KUKA KRL program: S_Zellenbereich.src, S_Zellenbereich.dat

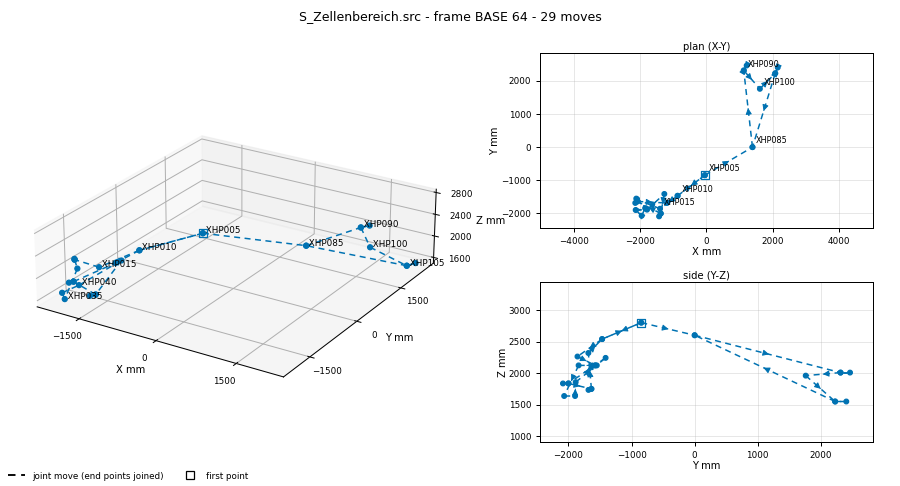
[picture p0: tool path of S_Zellenbereich.src in frame BASE 64, 29 of 31 moves have a stored position in this frame; points joined in program order, loops and branches not executed]
--- S_Zellenbereich.src ---
&ACCESS RVP
&REL 85
&COMMENT DAI_H_SOP_ZELLENBEREICH
&PARAM EDITMASK = DAI
&PARAM TEMPLATE = C:\KRC\roboter\template\vg_appl
&PARAM DISKPATH = KRC:\R1\H_Prog\DAI_SOP
DEF S_Zellenbereich( )
;FOLD INI;%{PE}
  ;FOLD BASISTECH INI
    GLOBAL INTERRUPT DECL 3 WHEN $STOPMESS==TRUE DO IR_STOPM ( )
    INTERRUPT ON 3
    BAS (#INITMOV,0 )
  ;ENDFOLD (BASISTECH INI)
  ;FOLD USER INI
    ;Make your modifications here
  ;ENDFOLD (USER INI)
;ENDFOLD (INI)
;FOLD ; Anlagenbezeichn: HC53_C    Stations-Nr: 060RB_100;%{PE}
;FOLD Parameters ;%{h}
;Params IlfProvider=kukaroboter.basistech.inlineforms.comments.comment; Kuka.Content=Anlagenbezeichn: HC53_C    Stations-Nr: 060RB_100
;ENDFOLD
;ENDFOLD
;FOLD ; Stand / Version: V1.0;%{PE}
;FOLD Parameters ;%{h}
;Params IlfProvider=kukaroboter.basistech.inlineforms.comments.comment; Kuka.Content=Stand / Version: V1.0
;ENDFOLD
;ENDFOLD
;FOLD ; Name Bearbeiter: EBZ-AE;%{PE}
;FOLD Parameters ;%{h}
;Params IlfProvider=kukaroboter.basistech.inlineforms.comments.comment; Kuka.Content=Name Bearbeiter: EBZ-AE
;ENDFOLD
;ENDFOLD
;FOLD ; Translator Version:29.01.2024 - Version 15.08;%{PE}
;FOLD Parameters ;%{h}
;Params IlfProvider=kukaroboter.basistech.inlineforms.comments.comment; Kuka.Content=Translator Version:29.01.2024 - Version 15.08
;ENDFOLD
;ENDFOLD

REPEAT
;FOLD MSG_T1
MSG_SHOW("DAI_H_SOP",#quit,999,"dai_h_sop_ok_0")
;ENDFOLD

; ***************************************
; A C H T U N G !!! Nur in $T1 abfahren
; ***************************************
UNTIL $T1 == TRUE

; ***************************************
; Pruefende Waende 4
;----------------------------------------
; Erreichbarkeit zum pruefen von P2/P3 nicht
; vorhanden.
;FOLD WAIT FOR ( IN 1026 'Vordefinierter Eingang immer ruckgesetzt.' )  ;%{PE}
;FOLD Parameters ;%{h}
;Params IlfProvider=kukaroboter.basistech.inlineforms.logics.waitfor; Kuka.WaitLogicTerm1=None; Kuka.WaitForNot1=False; Kuka.WaitLogicOp2.Term1=None; Kuka.WaitForNot2.Term1=False; Kuka.WaitForSysVar2.Term1=IN; Kuka.WaitForIndex2.Term1=1026; Kuka.WaitForIndexName2.Term1=Vordefinierter Eingang immer ruckgesetzt.; Kuka.WaitForTermNumbers=1; Kuka.WaitForOpNumbers=2; Kuka.WaitForCont=False
;ENDFOLD
WAIT FOR  ( $IN[1026] )
;ENDFOLD


;FOLD ; This program has been cleaned by KANERT_Makro. High risk of crash!!! Check the program carefully before deleting this comment. ;%{PE}
;FOLD Parameters ;%{h}
;Params IlfProvider=kukaroboter.basistech.inlineforms.comments.comment; Kuka.Content=This program has been cleaned by KANERT_Makro. High risk of crash!!! Check the program carefully before deleting this comment.
;ENDFOLD
WAIT FOR FALSE
;ENDFOLD
; ***************************************
;FOLD PTP HOME Vel=100 % DEFAULT;%{PE}
;FOLD Parameters ;%{h}
;Params IlfProvider=kukaroboter.basistech.inlineforms.movement.old; Kuka.IsGlobalPoint=False; Kuka.PointName=HOME; Kuka.BlendingEnabled=False; Kuka.MoveDataPtpName=DEFAULT; Kuka.VelocityPtp=100; Kuka.CurrentCDSetIndex=0; Kuka.MovementParameterFieldEnabled=True; IlfCommand=PTP
;ENDFOLD
$BWDSTART = FALSE
PDAT_ACT = PDEFAULT
FDAT_ACT = FHOME
BAS(#PTP_PARAMS, 100.0)
SET_CD_PARAMS (0)
PTP XHOME
;ENDFOLD

;Dynamische Pruefung Teil vorhanden
;FOLD PartPresent.CheckOff #1:5277, #2:5278, #3:1025, #4:1025, #5:1025, #6:1025, Bounce Time:100, Constant: Yes;%{PE}%
CheckPartPresent(5277,5278,1025,1025,1025,1025,100, True,FALSE)
;ENDFOLD

;Greifer-Ventile betatigen/pruefen
;FOLD DAI_GripValveCheck.Valve2 State:Fixierstift Ausfahren Gs, 060GRH101-QM1;%{PE}%
CheckValveState(2,1)
;ENDFOLD
;FOLD DAI_GripValveCheck.Valve3 State:Spanner Oeffnen Gs, 060GRH101-QM2;%{PE}%
CheckValveState(3,1)
;ENDFOLD
;FOLD DAI_GripValveCheck.Valve4 State:Spanner Oeffnen Gs, 060GRH101-QM3;%{PE}%
CheckValveState(4,1)
;ENDFOLD

;FOLD PTP HP005 Vel=100 % PDAT1 Tool[64]:Zero Base[64]:Zero ;%{PE}
;FOLD Parameters ;%{h}
;Params IlfProvider=kukaroboter.basistech.inlineforms.movement.old; Kuka.IsGlobalPoint=False; Kuka.PointName=HP005; Kuka.BlendingEnabled=False; Kuka.MoveDataPtpName=PDAT1; Kuka.VelocityPtp=100; Kuka.CurrentCDSetIndex=0; Kuka.MovementParameterFieldEnabled=True; IlfCommand=PTP
;ENDFOLD
$BWDSTART = FALSE
PDAT_ACT = PPDAT1
FDAT_ACT = FHP005
BAS(#PTP_PARAMS, 100.0)
SET_CD_PARAMS (0)
PTP XHP005
;ENDFOLD
;FOLD PTP HP010 Vel=100 % PDAT2 Tool[64]:Zero Base[64]:Zero ;%{PE}
;FOLD Parameters ;%{h}
;Params IlfProvider=kukaroboter.basistech.inlineforms.movement.old; Kuka.IsGlobalPoint=False; Kuka.PointName=HP010; Kuka.BlendingEnabled=False; Kuka.MoveDataPtpName=PDAT2; Kuka.VelocityPtp=100; Kuka.CurrentCDSetIndex=0; Kuka.MovementParameterFieldEnabled=True; IlfCommand=PTP
;ENDFOLD
$BWDSTART = FALSE
PDAT_ACT = PPDAT2
FDAT_ACT = FHP010
BAS(#PTP_PARAMS, 100.0)
SET_CD_PARAMS (0)
PTP XHP010
;ENDFOLD
;FOLD PTP HP015 Vel=100 % PDAT3 Tool[64]:Zero Base[64]:Zero ;%{PE}
;FOLD Parameters ;%{h}
;Params IlfProvider=kukaroboter.basistech.inlineforms.movement.old; Kuka.IsGlobalPoint=False; Kuka.PointName=HP015; Kuka.BlendingEnabled=False; Kuka.MoveDataPtpName=PDAT3; Kuka.VelocityPtp=100; Kuka.CurrentCDSetIndex=0; Kuka.MovementParameterFieldEnabled=True; IlfCommand=PTP
;ENDFOLD
$BWDSTART = FALSE
PDAT_ACT = PPDAT3
FDAT_ACT = FHP015
BAS(#PTP_PARAMS, 100.0)
SET_CD_PARAMS (0)
PTP XHP015
;ENDFOLD
;FOLD PTP HP020 Vel=100 % PDAT4 Tool[64]:Zero Base[64]:Zero;%{PE}
;FOLD Parameters ;%{h}
;Params IlfProvider=kukaroboter.basistech.inlineforms.movement.old; Kuka.IsGlobalPoint=False; Kuka.PointName=HP020; Kuka.BlendingEnabled=False; Kuka.MoveDataPtpName=PDAT4; Kuka.VelocityPtp=100; Kuka.CurrentCDSetIndex=0; Kuka.MovementParameterFieldEnabled=True; IlfCommand=PTP
;ENDFOLD
$BWDSTART = FALSE
PDAT_ACT = PPDAT4
FDAT_ACT = FHP020
BAS(#PTP_PARAMS, 100.0)
SET_CD_PARAMS (0)
PTP XHP020
;ENDFOLD

; Pruefung Raum P1n
;FOLD PTP LPruef01_Zellenbereich Vel=100 % PDAT5 Tool[64]:Zero Base[64]:Zero ;%{PE}
;FOLD Parameters ;%{h}
;Params IlfProvider=kukaroboter.basistech.inlineforms.movement.old; Kuka.IsGlobalPoint=False; Kuka.PointName=LPruef01_Zellenbereich; Kuka.BlendingEnabled=False; Kuka.MoveDataPtpName=PDAT5; Kuka.VelocityPtp=100; Kuka.CurrentCDSetIndex=0; Kuka.MovementParameterFieldEnabled=True; IlfCommand=PTP
;ENDFOLD
$BWDSTART = FALSE
PDAT_ACT = PPDAT5
FDAT_ACT = FLPruef01_Zellenbereich
BAS(#PTP_PARAMS, 100.0)
SET_CD_PARAMS (0)
PTP XLPruef01_Zellenbereich
;ENDFOLD
;FOLD PTP HP025 Vel=100 % PDAT6 Tool[64]:Zero Base[64]:Zero ;%{PE}
;FOLD Parameters ;%{h}
;Params IlfProvider=kukaroboter.basistech.inlineforms.movement.old; Kuka.IsGlobalPoint=False; Kuka.PointName=HP025; Kuka.BlendingEnabled=False; Kuka.MoveDataPtpName=PDAT6; Kuka.VelocityPtp=100; Kuka.CurrentCDSetIndex=0; Kuka.MovementParameterFieldEnabled=True; IlfCommand=PTP
;ENDFOLD
$BWDSTART = FALSE
PDAT_ACT = PPDAT6
FDAT_ACT = FHP025
BAS(#PTP_PARAMS, 100.0)
SET_CD_PARAMS (0)
PTP XHP025
;ENDFOLD
;FOLD PTP HP030 Vel=100 % PDAT7 Tool[64]:Zero Base[64]:Zero;%{PE}
;FOLD Parameters ;%{h}
;Params IlfProvider=kukaroboter.basistech.inlineforms.movement.old; Kuka.IsGlobalPoint=False; Kuka.PointName=HP030; Kuka.BlendingEnabled=False; Kuka.MoveDataPtpName=PDAT7; Kuka.VelocityPtp=100; Kuka.CurrentCDSetIndex=0; Kuka.MovementParameterFieldEnabled=True; IlfCommand=PTP
;ENDFOLD
$BWDSTART = FALSE
PDAT_ACT = PPDAT7
FDAT_ACT = FHP030
BAS(#PTP_PARAMS, 100.0)
SET_CD_PARAMS (0)
PTP XHP030
;ENDFOLD
;FOLD PTP HP035 Vel=100 % PDAT8 Tool[64]:Zero Base[64]:Zero;%{PE}
;FOLD Parameters ;%{h}
;Params IlfProvider=kukaroboter.basistech.inlineforms.movement.old; Kuka.IsGlobalPoint=False; Kuka.PointName=HP035; Kuka.BlendingEnabled=False; Kuka.MoveDataPtpName=PDAT8; Kuka.VelocityPtp=100; Kuka.CurrentCDSetIndex=0; Kuka.MovementParameterFieldEnabled=True; IlfCommand=PTP
;ENDFOLD
$BWDSTART = FALSE
PDAT_ACT = PPDAT8
FDAT_ACT = FHP035
BAS(#PTP_PARAMS, 100.0)
SET_CD_PARAMS (0)
PTP XHP035
;ENDFOLD

; Pruefung Raum P2
;FOLD PTP LPruef02_Zellenbereich Vel=100 % PDAT9 Tool[64]:Zero Base[64]:Zero ;%{PE}
;FOLD Parameters ;%{h}
;Params IlfProvider=kukaroboter.basistech.inlineforms.movement.old; Kuka.IsGlobalPoint=False; Kuka.PointName=LPruef02_Zellenbereich; Kuka.BlendingEnabled=False; Kuka.MoveDataPtpName=PDAT9; Kuka.VelocityPtp=100; Kuka.CurrentCDSetIndex=0; Kuka.MovementParameterFieldEnabled=True; IlfCommand=PTP
;ENDFOLD
$BWDSTART = FALSE
PDAT_ACT = PPDAT9
FDAT_ACT = FLPruef02_Zellenbereich
BAS(#PTP_PARAMS, 100.0)
SET_CD_PARAMS (0)
PTP XLPruef02_Zellenbereich
;ENDFOLD
;FOLD PTP HP040 Vel=100 % PDAT10 Tool[64]:Zero Base[64]:Zero ;%{PE}
;FOLD Parameters ;%{h}
;Params IlfProvider=kukaroboter.basistech.inlineforms.movement.old; Kuka.IsGlobalPoint=False; Kuka.PointName=HP040; Kuka.BlendingEnabled=False; Kuka.MoveDataPtpName=PDAT10; Kuka.VelocityPtp=100; Kuka.CurrentCDSetIndex=0; Kuka.MovementParameterFieldEnabled=True; IlfCommand=PTP
;ENDFOLD
$BWDSTART = FALSE
PDAT_ACT = PPDAT10
FDAT_ACT = FHP040
BAS(#PTP_PARAMS, 100.0)
SET_CD_PARAMS (0)
PTP XHP040
;ENDFOLD
;FOLD PTP HP045 Vel=100 % PDAT11 Tool[64]:Zero Base[64]:Zero ;%{PE}
;FOLD Parameters ;%{h}
;Params IlfProvider=kukaroboter.basistech.inlineforms.movement.old; Kuka.IsGlobalPoint=False; Kuka.PointName=HP045; Kuka.BlendingEnabled=False; Kuka.MoveDataPtpName=PDAT11; Kuka.VelocityPtp=100; Kuka.CurrentCDSetIndex=0; Kuka.MovementParameterFieldEnabled=True; IlfCommand=PTP
;ENDFOLD
$BWDSTART = FALSE
PDAT_ACT = PPDAT11
FDAT_ACT = FHP045
BAS(#PTP_PARAMS, 100.0)
SET_CD_PARAMS (0)
PTP XHP045
;ENDFOLD
;FOLD PTP HP050 Vel=100 % PDAT12 Tool[64]:Zero Base[64]:Zero ;%{PE}
;FOLD Parameters ;%{h}
;Params IlfProvider=kukaroboter.basistech.inlineforms.movement.old; Kuka.IsGlobalPoint=False; Kuka.PointName=HP050; Kuka.BlendingEnabled=False; Kuka.MoveDataPtpName=PDAT12; Kuka.VelocityPtp=100; Kuka.CurrentCDSetIndex=0; Kuka.MovementParameterFieldEnabled=True; IlfCommand=PTP
;ENDFOLD
$BWDSTART = FALSE
PDAT_ACT = PPDAT12
FDAT_ACT = FHP050
BAS(#PTP_PARAMS, 100.0)
SET_CD_PARAMS (0)
PTP XHP050
;ENDFOLD

; Pruefung Raum P3
;FOLD PTP LPruef03_Zellenbereich Vel=100 % PDAT13 Tool[64]:Zero Base[64]:Zero ;%{PE}
;FOLD Parameters ;%{h}
;Params IlfProvider=kukaroboter.basistech.inlineforms.movement.old; Kuka.IsGlobalPoint=False; Kuka.PointName=LPruef03_Zellenbereich; Kuka.BlendingEnabled=False; Kuka.MoveDataPtpName=PDAT13; Kuka.VelocityPtp=100; Kuka.CurrentCDSetIndex=0; Kuka.MovementParameterFieldEnabled=True; IlfCommand=PTP
;ENDFOLD
$BWDSTART = FALSE
PDAT_ACT = PPDAT13
FDAT_ACT = FLPruef03_Zellenbereich
BAS(#PTP_PARAMS, 100.0)
SET_CD_PARAMS (0)
PTP XLPruef03_Zellenbereich
;ENDFOLD
;FOLD PTP HP055 Vel=100 % PDAT14 Tool[64]:Zero Base[64]:Zero ;%{PE}
;FOLD Parameters ;%{h}
;Params IlfProvider=kukaroboter.basistech.inlineforms.movement.old; Kuka.IsGlobalPoint=False; Kuka.PointName=HP055; Kuka.BlendingEnabled=False; Kuka.MoveDataPtpName=PDAT14; Kuka.VelocityPtp=100; Kuka.CurrentCDSetIndex=0; Kuka.MovementParameterFieldEnabled=True; IlfCommand=PTP
;ENDFOLD
$BWDSTART = FALSE
PDAT_ACT = PPDAT14
FDAT_ACT = FHP055
BAS(#PTP_PARAMS, 100.0)
SET_CD_PARAMS (0)
PTP XHP055
;ENDFOLD
;FOLD PTP HP060 Vel=100 % PDAT15 Tool[64]:Zero Base[64]:Zero ;%{PE}
;FOLD Parameters ;%{h}
;Params IlfProvider=kukaroboter.basistech.inlineforms.movement.old; Kuka.IsGlobalPoint=False; Kuka.PointName=HP060; Kuka.BlendingEnabled=False; Kuka.MoveDataPtpName=PDAT15; Kuka.VelocityPtp=100; Kuka.CurrentCDSetIndex=0; Kuka.MovementParameterFieldEnabled=True; IlfCommand=PTP
;ENDFOLD
$BWDSTART = FALSE
PDAT_ACT = PPDAT15
FDAT_ACT = FHP060
BAS(#PTP_PARAMS, 100.0)
SET_CD_PARAMS (0)
PTP XHP060
;ENDFOLD

; Pruefung Raum P4
;FOLD PTP LPruef04_Zellenbereich Vel=100 % PDAT16 Tool[64]:Zero Base[64]:Zero ;%{PE}
;FOLD Parameters ;%{h}
;Params IlfProvider=kukaroboter.basistech.inlineforms.movement.old; Kuka.IsGlobalPoint=False; Kuka.PointName=LPruef04_Zellenbereich; Kuka.BlendingEnabled=False; Kuka.MoveDataPtpName=PDAT16; Kuka.VelocityPtp=100; Kuka.CurrentCDSetIndex=0; Kuka.MovementParameterFieldEnabled=True; IlfCommand=PTP
;ENDFOLD
$BWDSTART = FALSE
PDAT_ACT = PPDAT16
FDAT_ACT = FLPruef04_Zellenbereich
BAS(#PTP_PARAMS, 100.0)
SET_CD_PARAMS (0)
PTP XLPruef04_Zellenbereich
;ENDFOLD
;FOLD PTP HP065 Vel=100 % PDAT17 Tool[64]:Zero Base[64]:Zero ;%{PE}
;FOLD Parameters ;%{h}
;Params IlfProvider=kukaroboter.basistech.inlineforms.movement.old; Kuka.IsGlobalPoint=False; Kuka.PointName=HP065; Kuka.BlendingEnabled=False; Kuka.MoveDataPtpName=PDAT17; Kuka.VelocityPtp=100; Kuka.CurrentCDSetIndex=0; Kuka.MovementParameterFieldEnabled=True; IlfCommand=PTP
;ENDFOLD
$BWDSTART = FALSE
PDAT_ACT = PPDAT17
FDAT_ACT = FHP065
BAS(#PTP_PARAMS, 100.0)
SET_CD_PARAMS (0)
PTP XHP065
;ENDFOLD
;FOLD PTP HP070 Vel=100 % PDAT18 Tool[64]:Zero Base[64]:Zero ;%{PE}
;FOLD Parameters ;%{h}
;Params IlfProvider=kukaroboter.basistech.inlineforms.movement.old; Kuka.IsGlobalPoint=False; Kuka.PointName=HP070; Kuka.BlendingEnabled=False; Kuka.MoveDataPtpName=PDAT18; Kuka.VelocityPtp=100; Kuka.CurrentCDSetIndex=0; Kuka.MovementParameterFieldEnabled=True; IlfCommand=PTP
;ENDFOLD
$BWDSTART = FALSE
PDAT_ACT = PPDAT18
FDAT_ACT = FHP070
BAS(#PTP_PARAMS, 100.0)
SET_CD_PARAMS (0)
PTP XHP070
;ENDFOLD
;FOLD PTP HP075 Vel=100 % PDAT19 Tool[64]:Zero Base[64]:Zero ;%{PE}
;FOLD Parameters ;%{h}
;Params IlfProvider=kukaroboter.basistech.inlineforms.movement.old; Kuka.IsGlobalPoint=False; Kuka.PointName=HP075; Kuka.BlendingEnabled=False; Kuka.MoveDataPtpName=PDAT19; Kuka.VelocityPtp=100; Kuka.CurrentCDSetIndex=0; Kuka.MovementParameterFieldEnabled=True; IlfCommand=PTP
;ENDFOLD
$BWDSTART = FALSE
PDAT_ACT = PPDAT19
FDAT_ACT = FHP075
BAS(#PTP_PARAMS, 100.0)
SET_CD_PARAMS (0)
PTP XHP075
;ENDFOLD
;FOLD PTP HP080 Vel=100 % PDAT20 Tool[64]:Zero Base[64]:Zero ;%{PE}
;FOLD Parameters ;%{h}
;Params IlfProvider=kukaroboter.basistech.inlineforms.movement.old; Kuka.IsGlobalPoint=False; Kuka.PointName=HP080; Kuka.BlendingEnabled=False; Kuka.MoveDataPtpName=PDAT20; Kuka.VelocityPtp=100; Kuka.CurrentCDSetIndex=0; Kuka.MovementParameterFieldEnabled=True; IlfCommand=PTP
;ENDFOLD
$BWDSTART = FALSE
PDAT_ACT = PPDAT20
FDAT_ACT = FHP080
BAS(#PTP_PARAMS, 100.0)
SET_CD_PARAMS (0)
PTP XHP080
;ENDFOLD
;FOLD PTP HP085 Vel=100 % PDAT21 Tool[64]:Zero Base[64]:Zero ;%{PE}
;FOLD Parameters ;%{h}
;Params IlfProvider=kukaroboter.basistech.inlineforms.movement.old; Kuka.IsGlobalPoint=False; Kuka.PointName=HP085; Kuka.BlendingEnabled=False; Kuka.MoveDataPtpName=PDAT21; Kuka.VelocityPtp=100; Kuka.CurrentCDSetIndex=0; Kuka.MovementParameterFieldEnabled=True; IlfCommand=PTP
;ENDFOLD
$BWDSTART = FALSE
PDAT_ACT = PPDAT21
FDAT_ACT = FHP085
BAS(#PTP_PARAMS, 100.0)
SET_CD_PARAMS (0)
PTP XHP085
;ENDFOLD
;FOLD PTP HP090 Vel=100 % PDAT22 Tool[64]:Zero Base[64]:Zero;%{PE}
;FOLD Parameters ;%{h}
;Params IlfProvider=kukaroboter.basistech.inlineforms.movement.old; Kuka.IsGlobalPoint=False; Kuka.PointName=HP090; Kuka.BlendingEnabled=False; Kuka.MoveDataPtpName=PDAT22; Kuka.VelocityPtp=100; Kuka.CurrentCDSetIndex=0; Kuka.MovementParameterFieldEnabled=True; IlfCommand=PTP
;ENDFOLD
$BWDSTART = FALSE
PDAT_ACT = PPDAT22
FDAT_ACT = FHP090
BAS(#PTP_PARAMS, 100.0)
SET_CD_PARAMS (0)
PTP XHP090
;ENDFOLD

; Pruefung Raum P5
;FOLD PTP LPruef05_Zellenbereich Vel=100 % PDAT23 Tool[64]:Zero Base[64]:Zero ;%{PE}
;FOLD Parameters ;%{h}
;Params IlfProvider=kukaroboter.basistech.inlineforms.movement.old; Kuka.IsGlobalPoint=False; Kuka.PointName=LPruef05_Zellenbereich; Kuka.BlendingEnabled=False; Kuka.MoveDataPtpName=PDAT23; Kuka.VelocityPtp=100; Kuka.CurrentCDSetIndex=0; Kuka.MovementParameterFieldEnabled=True; IlfCommand=PTP
;ENDFOLD
$BWDSTART = FALSE
PDAT_ACT = PPDAT23
FDAT_ACT = FLPruef05_Zellenbereich
BAS(#PTP_PARAMS, 100.0)
SET_CD_PARAMS (0)
PTP XLPruef05_Zellenbereich
;ENDFOLD
;FOLD PTP HP095 Vel=100 % PDAT24 Tool[64]:Zero Base[64]:Zero ;%{PE}
;FOLD Parameters ;%{h}
;Params IlfProvider=kukaroboter.basistech.inlineforms.movement.old; Kuka.IsGlobalPoint=False; Kuka.PointName=HP095; Kuka.BlendingEnabled=False; Kuka.MoveDataPtpName=PDAT24; Kuka.VelocityPtp=100; Kuka.CurrentCDSetIndex=0; Kuka.MovementParameterFieldEnabled=True; IlfCommand=PTP
;ENDFOLD
$BWDSTART = FALSE
PDAT_ACT = PPDAT24
FDAT_ACT = FHP095
BAS(#PTP_PARAMS, 100.0)
SET_CD_PARAMS (0)
PTP XHP095
;ENDFOLD
;FOLD PTP HP100 Vel=100 % PDAT25 Tool[64]:Zero Base[64]:Zero;%{PE}
;FOLD Parameters ;%{h}
;Params IlfProvider=kukaroboter.basistech.inlineforms.movement.old; Kuka.IsGlobalPoint=False; Kuka.PointName=HP100; Kuka.BlendingEnabled=False; Kuka.MoveDataPtpName=PDAT25; Kuka.VelocityPtp=100; Kuka.CurrentCDSetIndex=0; Kuka.MovementParameterFieldEnabled=True; IlfCommand=PTP
;ENDFOLD
$BWDSTART = FALSE
PDAT_ACT = PPDAT25
FDAT_ACT = FHP100
BAS(#PTP_PARAMS, 100.0)
SET_CD_PARAMS (0)
PTP XHP100
;ENDFOLD
;FOLD PTP HP105 Vel=100 % PDAT26 Tool[64]:Zero Base[64]:Zero;%{PE}
;FOLD Parameters ;%{h}
;Params IlfProvider=kukaroboter.basistech.inlineforms.movement.old; Kuka.IsGlobalPoint=False; Kuka.PointName=HP105; Kuka.BlendingEnabled=False; Kuka.MoveDataPtpName=PDAT26; Kuka.VelocityPtp=100; Kuka.CurrentCDSetIndex=0; Kuka.MovementParameterFieldEnabled=True; IlfCommand=PTP
;ENDFOLD
$BWDSTART = FALSE
PDAT_ACT = PPDAT26
FDAT_ACT = FHP105
BAS(#PTP_PARAMS, 100.0)
SET_CD_PARAMS (0)
PTP XHP105
;ENDFOLD

; Pruefung Raum P6
;FOLD PTP LPruef06_Zellenbereich Vel=100 % PDAT27 Tool[64]:Zero Base[64]:Zero ;%{PE}
;FOLD Parameters ;%{h}
;Params IlfProvider=kukaroboter.basistech.inlineforms.movement.old; Kuka.IsGlobalPoint=False; Kuka.PointName=LPruef06_Zellenbereich; Kuka.BlendingEnabled=False; Kuka.MoveDataPtpName=PDAT27; Kuka.VelocityPtp=100; Kuka.CurrentCDSetIndex=0; Kuka.MovementParameterFieldEnabled=True; IlfCommand=PTP
;ENDFOLD
$BWDSTART = FALSE
PDAT_ACT = PPDAT27
FDAT_ACT = FLPruef06_Zellenbereich
BAS(#PTP_PARAMS, 100.0)
SET_CD_PARAMS (0)
PTP XLPruef06_Zellenbereich
;ENDFOLD
;FOLD PTP HP110 Vel=100 % PDAT28 Tool[64]:Zero Base[64]:Zero;%{PE}
;FOLD Parameters ;%{h}
;Params IlfProvider=kukaroboter.basistech.inlineforms.movement.old; Kuka.IsGlobalPoint=False; Kuka.PointName=HP110; Kuka.BlendingEnabled=False; Kuka.MoveDataPtpName=PDAT28; Kuka.VelocityPtp=100; Kuka.CurrentCDSetIndex=0; Kuka.MovementParameterFieldEnabled=True; IlfCommand=PTP
;ENDFOLD
$BWDSTART = FALSE
PDAT_ACT = PPDAT28
FDAT_ACT = FHP110
BAS(#PTP_PARAMS, 100.0)
SET_CD_PARAMS (0)
PTP XHP110
;ENDFOLD
;FOLD PTP HP115 Vel=100 % PDAT29 Tool[64]:Zero Base[64]:Zero;%{PE}
;FOLD Parameters ;%{h}
;Params IlfProvider=kukaroboter.basistech.inlineforms.movement.old; Kuka.IsGlobalPoint=False; Kuka.PointName=HP115; Kuka.BlendingEnabled=False; Kuka.MoveDataPtpName=PDAT29; Kuka.VelocityPtp=100; Kuka.CurrentCDSetIndex=0; Kuka.MovementParameterFieldEnabled=True; IlfCommand=PTP
;ENDFOLD
$BWDSTART = FALSE
PDAT_ACT = PPDAT29
FDAT_ACT = FHP115
BAS(#PTP_PARAMS, 100.0)
SET_CD_PARAMS (0)
PTP XHP115
;ENDFOLD

;FOLD PTP HOME Vel=100 % DEFAULT;%{PE}
;FOLD Parameters ;%{h}
;Params IlfProvider=kukaroboter.basistech.inlineforms.movement.old; Kuka.IsGlobalPoint=False; Kuka.PointName=HOME; Kuka.BlendingEnabled=False; Kuka.MoveDataPtpName=DEFAULT; Kuka.VelocityPtp=100; Kuka.CurrentCDSetIndex=0; Kuka.MovementParameterFieldEnabled=True; IlfCommand=PTP
;ENDFOLD
$BWDSTART = FALSE
PDAT_ACT = PDEFAULT
FDAT_ACT = FHOME
BAS(#PTP_PARAMS, 100.0)
SET_CD_PARAMS (0)
PTP XHOME
;ENDFOLD

;Collision detection - Off
;FOLD COLLDETECT Off ;%{PE}
;FOLD Parameters ;%{h}
;Params IlfProvider=kukaroboter.basistech.inlineforms.colldetect.off; CollDetect.Command=Off
;ENDFOLD
USE_CD_PARAMS(0)
;ENDFOLD
END

--- S_Zellenbereich.dat ---
&ACCESS RVO
&REL 86
&COMMENT DAI_H_SOP_ZELLENBEREICH
&PARAM EDITMASK = DAI
&PARAM TEMPLATE = C:\KRC\roboter\template\vg_appl
&PARAM DISKPATH = KRC:\R1\H_Prog\DAI_SOP
DEFDAT  S_ZELLENBEREICH
;FOLD EXTERNAL DECLARATIONS;%{PE}%MKUKATPBASIS,%CEXT,%VCOMMON,%P
;FOLD BASISTECH EXT;%{PE}%MKUKATPBASIS,%CEXT,%VEXT,%P
EXT  BAS (BAS_COMMAND  :IN,REAL  :IN )
DECL INT SUCCESS
;ENDFOLD (BASISTECH EXT)
;FOLD USER EXT;%{E}%MKUKATPUSER,%CEXT,%VEXT,%P
;Make your modifications here
;ENDFOLD (USER EXT)
;FOLD COLLISION
EXT  COLLSTOP (INT  :IN,INT  :IN )
;ENDFOLD  (Collision)
;ENDFOLD (EXTERNAL DECLERATIONS)
DECL BASIS_SUGG_T LAST_BASIS={POINT1[] "P0                      ",POINT2[] "P0                      ",CP_PARAMS[] "CPDAT0                  ",PTP_PARAMS[] "PDAT0                   ",CONT[] "                        ",CP_VEL[] "2.0                     ",PTP_VEL[] "100                     ",SYNC_PARAMS[] "SYNCDAT                 ",SPL_NAME[] "S0                      ",A_PARAMS[] "ADAT0                   "}
DECL MODULEPARAM_T LAST_TP_PARAMS={PARAMS[] "Kuka.PointName=LPruef11_Zellenbereich; Kuka.FrameData.base_no=64; Kuka.FrameData.tool_no=64; Kuka.FrameData.ipo_frame=#BASE; Kuka.FrameData.point2=; Kuka.isglobalpoint=False; Kuka.MoveDataPtpName=PDAT42; Kuka.MovementDataPdat.apo_mode=#CDIS; Kuka.MovementDataPdat.apo_dist=500; Kuka.MovementData.vel=100; Kuka.MovementData.acc=100; Kuka.MovementData.exax_ign=0; Kuka.VelocityPtp=100; Kuka.BlendingEnabled=False; Kuka.APXEnabled=False; Kuka.CurrentCDSetIndex=0"}

; E6POS Declarations
DECL E6POS XHP005={X -46.1297722,Y -846.191040,Z 2801.22607,A 172.487946,B -23.7688217,C -126.323227,S 18,T 10,E1 -351.691864,E2 0.0,E3 0.0,E4 0.0,E5 0.0,E6 0.0}
DECL E6POS XHP010={X -867.191101,Y -1466.68518,Z 2540.40723,A -152.699829,B -31.1417503,C -161.784149,S 18,T 10,E1 -164.100861,E2 0.0,E3 0.0,E4 0.0,E5 0.0,E6 0.0}
DECL E6POS XHP015={X -1396.02393,Y -1857.07593,Z 2264.14600,A -150.484390,B -25.5367279,C -163.976059,S 18,T 10,E1 21.3274384,E2 0.0,E3 0.0,E4 0.0,E5 0.0,E6 0.0}
DECL E6POS XHP020={X -2092.19604,Y -1575.54126,Z 2123.50146,A 154.259888,B -12.4955034,C -157.719711,S 18,T 2,E1 139.994904,E2 0.0,E3 0.0,E4 0.0,E5 0.0,E6 0.0}
DECL E6POS XLPruef01_Zellenbereich={X -2113.71436,Y -1551.14844,Z 2123.29077,A 154.254562,B -12.4912186,C -157.727356,S 18,T 2,E1 139.979416,E2 0.0,E3 0.0,E4 0.0,E5 0.0,E6 0.0}
DECL E6POS XHP025={X -2092.19604,Y -1575.54126,Z 2123.50146,A 154.259888,B -12.4955034,C -157.719711,S 18,T 2,E1 139.994904,E2 0.0,E3 0.0,E4 0.0,E5 0.0,E6 0.0}
DECL E6POS XHP030={X -1845.86414,Y -1839.41907,Z 2123.51465,A 162.511520,B -12.4958191,C -157.719528,S 18,T 2,E1 139.994904,E2 0.0,E3 0.0,E4 0.0,E5 0.0,E6 0.0}
DECL E6POS XHP035={X -1951.68848,Y -2068.02368,Z 1638.32666,A -82.6358185,B -21.5607433,C 152.311325,S 18,T 2,E1 138.383224,E2 0.0,E3 0.0,E4 0.0,E5 0.0,E6 0.0}
DECL E6POS XLPruef02_Zellenbereich={X -2131.54565,Y -1895.27588,Z 1638.31763,A -87.8327,B -21.5607204,C 152.311584,S 18,T 2,E1 138.383224,E2 0.0,E3 0.0,E4 0.0,E5 0.0,E6 0.0}
DECL E6POS XHP040={X -1789.18262,Y -1885.51208,Z 1857.81531,A -81.9620132,B -20.7954330,C 153.753494,S 18,T 2,E1 137.819962,E2 0.0,E3 0.0,E4 0.0,E5 0.0,E6 0.0}
DECL E6POS XHP045={X -1267.41907,Y -1411.34326,Z 2242.63013,A -22.7016411,B -28.9057846,C 101.976242,S 18,T 10,E1 100.000,E2 0.0,E3 0.0,E4 0.0,E5 0.0,E6 0.0}
DECL E6POS XHP050={X -1375.15015,Y -2000.49536,Z 1837.26526,A -20.9162292,B -32.2844200,C 114.147118,S 18,T 10,E1 100.000,E2 0.0,E3 0.0,E4 0.0,E5 0.0,E6 0.0}
DECL E6POS XLPruef03_Zellenbereich={X -1425.14453,Y -2087.10596,Z 1837.26392,A -20.9162064,B -32.2844238,C 114.147110,S 18,T 10,E1 100.000,E2 0.0,E3 0.0,E4 0.0,E5 0.0,E6 0.0}
DECL E6POS XHP055={X -1375.15430,Y -2000.50244,Z 1837.26221,A -20.9162197,B -32.2844276,C 114.147110,S 18,T 10,E1 100.000,E2 0.0,E3 0.0,E4 0.0,E5 0.0,E6 0.0}
DECL E6POS XHP060={X -2083.14478,Y -1636.46228,Z 1751.08667,A -63.3908806,B -28.3927116,C 157.657501,S 18,T 10,E1 100.002556,E2 0.0,E3 0.0,E4 0.0,E5 0.0,E6 0.0}
DECL E6POS XLPruef04_Zellenbereich={X -2144.09473,Y -1682.65088,Z 1735.18335,A -61.9271507,B -28.8603210,C 154.600876,S 18,T 10,E1 100.002556,E2 0.0,E3 0.0,E4 0.0,E5 0.0,E6 0.0}
DECL E6POS XHP065={X -2083.14478,Y -1636.46228,Z 1751.08667,A -63.3908806,B -28.3927116,C 157.657501,S 18,T 10,E1 100.002556,E2 0.0,E3 0.0,E4 0.0,E5 0.0,E6 0.0}
DECL E6POS XHP070={X -1191.14673,Y -1684.66479,Z 2320.02466,A -116.427757,B -34.0038147,C -176.647430,S 18,T 10,E1 -72.8242340,E2 0.0,E3 0.0,E4 0.0,E5 0.0,E6 0.0}
DECL E6POS XHP075={X -867.191101,Y -1466.68518,Z 2540.40723,A -152.699829,B -31.1417503,C -161.784149,S 18,T 10,E1 -164.100861,E2 0.0,E3 0.0,E4 0.0,E5 0.0,E6 0.0}
DECL E6POS XHP080={X -46.1297722,Y -846.191040,Z 2801.22607,A 172.487946,B -23.7688217,C -126.323227,S 18,T 10,E1 -351.691864,E2 0.0,E3 0.0,E4 0.0,E5 0.0,E6 0.0}
DECL E6POS XHP085={X 1391.85376,Y 0.356020540,Z 2601.24731,A -90.0283508,B -0.0163251683,C -129.966507,S 18,T 11,E1 -500.000,E2 0.0,E3 0.0,E4 0.0,E5 0.0,E6 0.0}
DECL E6POS XHP090={X 1129.05261,Y 2312.21265,Z 2009.50732,A -12.2057838,B -168.133545,C -51.1410065,S 18,T 11,E1 -500.000,E2 0.0,E3 0.0,E4 0.0,E5 0.0,E6 0.0}
DECL E6POS XLPruef05_Zellenbereich={X 1216.39185,Y 2462.71387,Z 2009.50720,A -12.2057009,B -168.133545,C -51.1410370,S 18,T 11,E1 -500.000,E2 0.0,E3 0.0,E4 0.0,E5 0.0,E6 0.0}
DECL E6POS XHP095={X 1129.05493,Y 2312.22046,Z 2009.50659,A -12.2057762,B -168.133530,C -51.1410141,S 18,T 11,E1 -500.000,E2 0.0,E3 0.0,E4 0.0,E5 0.0,E6 0.0}
DECL E6POS XHP100={X 1614.92224,Y 1760.35242,Z 1961.21033,A -18.5538177,B 13.2130013,C -144.386597,S 18,T 11,E1 -500.000183,E2 0.0,E3 0.0,E4 0.0,E5 0.0,E6 0.0}
DECL E6POS XHP105={X 2078.72,Y 2226.96118,Z 1551.24170,A -27.8164654,B 5.86191130,C -111.963608,S 18,T 11,E1 -500.012482,E2 0.0,E3 0.0,E4 0.0,E5 0.0,E6 0.0}
DECL E6POS XLPruef06_Zellenbereich={X 2153.80737,Y 2403.58984,Z 1551.19421,A -27.8202477,B 5.86857748,C -111.963539,S 18,T 11,E1 -500.012695,E2 0.0,E3 0.0,E4 0.0,E5 0.0,E6 0.0}
DECL E6POS XHP110={X 2078.72,Y 2226.96118,Z 1551.24170,A -27.8164692,B 5.86191,C -111.963615,S 18,T 11,E1 -500.012482,E2 0.0,E3 0.0,E4 0.0,E5 0.0,E6 0.0}
DECL E6POS XHP115={X 1391.85376,Y 0.356020540,Z 2601.24731,A -90.0283508,B -0.0163251683,C -129.966507,S 18,T 10,E1 -500.000,E2 0.0,E3 0.0,E4 0.0,E5 0.0,E6 0.0}

; PDAT/LDAT Declarations
DECL PDAT PPDAT1={VEL 100.000,ACC 100.000,APO_DIST 500.000,APO_MODE #CDIS,GEAR_JERK 100.000,EXAX_IGN 0}
DECL PDAT PPDAT2={VEL 100.000,ACC 100.000,APO_DIST 500.000,APO_MODE #CDIS,GEAR_JERK 100.000,EXAX_IGN 0}
DECL PDAT PPDAT3={VEL 100.000,ACC 100.000,APO_DIST 500.000,APO_MODE #CDIS,GEAR_JERK 100.000,EXAX_IGN 0}
DECL PDAT PPDAT4={VEL 100.000,ACC 100.000,APO_DIST 0.0,APO_MODE #CDIS,GEAR_JERK 50.0000,EXAX_IGN 0}
DECL PDAT PPDAT5={VEL 100.000,ACC 100.000,APO_DIST 500.000,APO_MODE #CDIS,GEAR_JERK 100.000,EXAX_IGN 0}
DECL PDAT PPDAT6={VEL 100.000,ACC 100.000,APO_DIST 500.000,APO_MODE #CDIS,GEAR_JERK 100.000,EXAX_IGN 0}
DECL PDAT PPDAT7={VEL 100.000,ACC 100.000,APO_DIST 0.0,APO_MODE #CDIS,GEAR_JERK 50.0000,EXAX_IGN 0}
DECL PDAT PPDAT8={VEL 100.000,ACC 100.000,APO_DIST 0.0,APO_MODE #CDIS,GEAR_JERK 50.0000,EXAX_IGN 0}
DECL PDAT PPDAT9={VEL 100.000,ACC 100.000,APO_DIST 500.000,APO_MODE #CDIS,GEAR_JERK 100.000,EXAX_IGN 0}
DECL PDAT PPDAT10={VEL 100.000,ACC 100.000,APO_DIST 0.0,APO_MODE #CDIS,GEAR_JERK 50.0000,EXAX_IGN 0}
DECL PDAT PPDAT11={VEL 100.000,ACC 100.000,APO_DIST 0.0,APO_MODE #CDIS,GEAR_JERK 50.0000,EXAX_IGN 0}
DECL PDAT PPDAT12={VEL 100.000,ACC 100.000,APO_DIST 0.0,APO_MODE #CDIS,GEAR_JERK 50.0000,EXAX_IGN 0}
DECL PDAT PPDAT13={VEL 100.000,ACC 100.000,APO_DIST 500.000,APO_MODE #CDIS,GEAR_JERK 100.000,EXAX_IGN 0}
DECL PDAT PPDAT14={VEL 100.000,ACC 100.000,APO_DIST 500.000,APO_MODE #CDIS,GEAR_JERK 100.000,EXAX_IGN 0}
DECL PDAT PPDAT15={VEL 100.000,ACC 100.000,APO_DIST 0.0,APO_MODE #CDIS,GEAR_JERK 50.0000,EXAX_IGN 0}
DECL PDAT PPDAT16={VEL 100.000,ACC 100.000,APO_DIST 500.000,APO_MODE #CDIS,GEAR_JERK 100.000,EXAX_IGN 0}
DECL PDAT PPDAT17={VEL 100.000,ACC 100.000,APO_DIST 500.000,APO_MODE #CDIS,GEAR_JERK 100.000,EXAX_IGN 0}
DECL PDAT PPDAT18={VEL 100.000,ACC 100.000,APO_DIST 500.000,APO_MODE #CDIS,GEAR_JERK 100.000,EXAX_IGN 0}
DECL PDAT PPDAT19={VEL 100.000,ACC 100.000,APO_DIST 0.0,APO_MODE #CDIS,GEAR_JERK 50.0000,EXAX_IGN 0}
DECL PDAT PPDAT20={VEL 100.000,ACC 100.000,APO_DIST 500.000,APO_MODE #CDIS,GEAR_JERK 100.000,EXAX_IGN 0}
DECL PDAT PPDAT21={VEL 100.000,ACC 100.000,APO_DIST 500.000,APO_MODE #CDIS,GEAR_JERK 100.000,EXAX_IGN 0}
DECL PDAT PPDAT22={VEL 100.000,ACC 100.000,APO_DIST 0.0,APO_MODE #CDIS,GEAR_JERK 50.0000,EXAX_IGN 0}
DECL PDAT PPDAT23={VEL 100.000,ACC 100.000,APO_DIST 500.000,APO_MODE #CDIS,GEAR_JERK 100.000,EXAX_IGN 0}
DECL PDAT PPDAT24={VEL 100.000,ACC 100.000,APO_DIST 500.000,APO_MODE #CDIS,GEAR_JERK 100.000,EXAX_IGN 0}
DECL PDAT PPDAT25={VEL 100.000,ACC 100.000,APO_DIST 0.0,APO_MODE #CDIS,GEAR_JERK 50.0000,EXAX_IGN 0}
DECL PDAT PPDAT26={VEL 100.000,ACC 100.000,APO_DIST 0.0,APO_MODE #CDIS,GEAR_JERK 50.0000,EXAX_IGN 0}
DECL PDAT PPDAT27={VEL 100.000,ACC 100.000,APO_DIST 500.000,APO_MODE #CDIS,GEAR_JERK 100.000,EXAX_IGN 0}
DECL PDAT PPDAT28={VEL 100.000,ACC 100.000,APO_DIST 0.0,APO_MODE #CDIS,GEAR_JERK 50.0000,EXAX_IGN 0}
DECL PDAT PPDAT29={VEL 100.000,ACC 100.000,APO_DIST 0.0,APO_MODE #CDIS,GEAR_JERK 50.0000,EXAX_IGN 0}

; FDAT Declarations
DECL FDAT FHOME={TOOL_NO 64,BASE_NO 64,IPO_FRAME #BASE,POINT2[] " "}
DECL FDAT FHP005={TOOL_NO 64,BASE_NO 64,IPO_FRAME #BASE,POINT2[] " "}
DECL FDAT FHP010={TOOL_NO 64,BASE_NO 64,IPO_FRAME #BASE,POINT2[] " "}
DECL FDAT FHP015={TOOL_NO 64,BASE_NO 64,IPO_FRAME #BASE,POINT2[] " "}
DECL FDAT FHP020={TOOL_NO 64,BASE_NO 64,IPO_FRAME #BASE,POINT2[] " "}
DECL FDAT FLPruef01_Zellenbereich={TOOL_NO 64,BASE_NO 64,IPO_FRAME #BASE,POINT2[] " "}
DECL FDAT FHP025={TOOL_NO 64,BASE_NO 64,IPO_FRAME #BASE,POINT2[] " "}
DECL FDAT FHP030={TOOL_NO 64,BASE_NO 64,IPO_FRAME #BASE,POINT2[] " "}
DECL FDAT FHP035={TOOL_NO 64,BASE_NO 64,IPO_FRAME #BASE,POINT2[] " "}
DECL FDAT FLPruef02_Zellenbereich={TOOL_NO 64,BASE_NO 64,IPO_FRAME #BASE,POINT2[] " "}
DECL FDAT FHP040={TOOL_NO 64,BASE_NO 64,IPO_FRAME #BASE,POINT2[] " "}
DECL FDAT FHP045={TOOL_NO 64,BASE_NO 64,IPO_FRAME #BASE,POINT2[] " "}
DECL FDAT FHP050={TOOL_NO 64,BASE_NO 64,IPO_FRAME #BASE,POINT2[] " "}
DECL FDAT FLPruef03_Zellenbereich={TOOL_NO 64,BASE_NO 64,IPO_FRAME #BASE,POINT2[] " "}
DECL FDAT FHP055={TOOL_NO 64,BASE_NO 64,IPO_FRAME #BASE,POINT2[] " "}
DECL FDAT FHP060={TOOL_NO 64,BASE_NO 64,IPO_FRAME #BASE,POINT2[] " "}
DECL FDAT FLPruef04_Zellenbereich={TOOL_NO 64,BASE_NO 64,IPO_FRAME #BASE,POINT2[] " "}
DECL FDAT FHP065={TOOL_NO 64,BASE_NO 64,IPO_FRAME #BASE,POINT2[] " "}
DECL FDAT FHP070={TOOL_NO 64,BASE_NO 64,IPO_FRAME #BASE,POINT2[] " "}
DECL FDAT FHP075={TOOL_NO 64,BASE_NO 64,IPO_FRAME #BASE,POINT2[] " "}
DECL FDAT FHP080={TOOL_NO 64,BASE_NO 64,IPO_FRAME #BASE,POINT2[] " "}
DECL FDAT FHP085={TOOL_NO 64,BASE_NO 64,IPO_FRAME #BASE,POINT2[] " "}
DECL FDAT FHP090={TOOL_NO 64,BASE_NO 64,IPO_FRAME #BASE,POINT2[] " "}
DECL FDAT FLPruef05_Zellenbereich={TOOL_NO 64,BASE_NO 64,IPO_FRAME #BASE,POINT2[] " "}
DECL FDAT FHP095={TOOL_NO 64,BASE_NO 64,IPO_FRAME #BASE,POINT2[] " "}
DECL FDAT FHP100={TOOL_NO 64,BASE_NO 64,IPO_FRAME #BASE,POINT2[] " "}
DECL FDAT FHP105={TOOL_NO 64,BASE_NO 64,IPO_FRAME #BASE,POINT2[] " "}
DECL FDAT FLPruef06_Zellenbereich={TOOL_NO 64,BASE_NO 64,IPO_FRAME #BASE,POINT2[] " "}
DECL FDAT FHP110={TOOL_NO 64,BASE_NO 64,IPO_FRAME #BASE,POINT2[] " "}
DECL FDAT FHP115={TOOL_NO 64,BASE_NO 64,IPO_FRAME #BASE,POINT2[] " "}

ENDDAT
